FUNCTION_BLOCK FB_Carro_GRF_LD
// Transcripción del grafcet (GRF -> LD) [Usando células eléctricas de memoria]
VAR_INPUT
    ManiobrasTotales: UINT := 2;
    TiempoEspera: TIME := T#2S;
END_VAR
VAR_OUTPUT
    ManiobrasPendientes: UINT;
    TiempoPendiente: TIME;
END_VAR
VAR
    TiempoActual: TIME;
    
    // Variables propias del GRF
    S0x: BOOL := TRUE; // Etapa inicial
    S1x, S2x, S3x, S4x: BOOL; // Etapas no-iniciales
    t0, t1, t2, t3, t4, t4a: BOOL; // Transiciones
    S2t, S2_t: TIME; // S2.t y S2._t
    
    // Bloques funcionales
    FlancoPulsadorMarcha: R_TRIG;
    Intermitencia: FB_Blink;
    
    // Entradas
    i_PulsadorMarcha AT %I*: BOOL;
    i_FinalCarreraIzquierda AT %I*: BOOL := TRUE;
    i_FinalCarreraDerecha AT %I*: BOOL;
    
    // Salidas
    o_MarchaIzquierda AT %I*: BOOL;
    o_MarchaDerecha AT %I*: BOOL;
    o_LamparaMarcha AT %I*: BOOL;
END_VAR

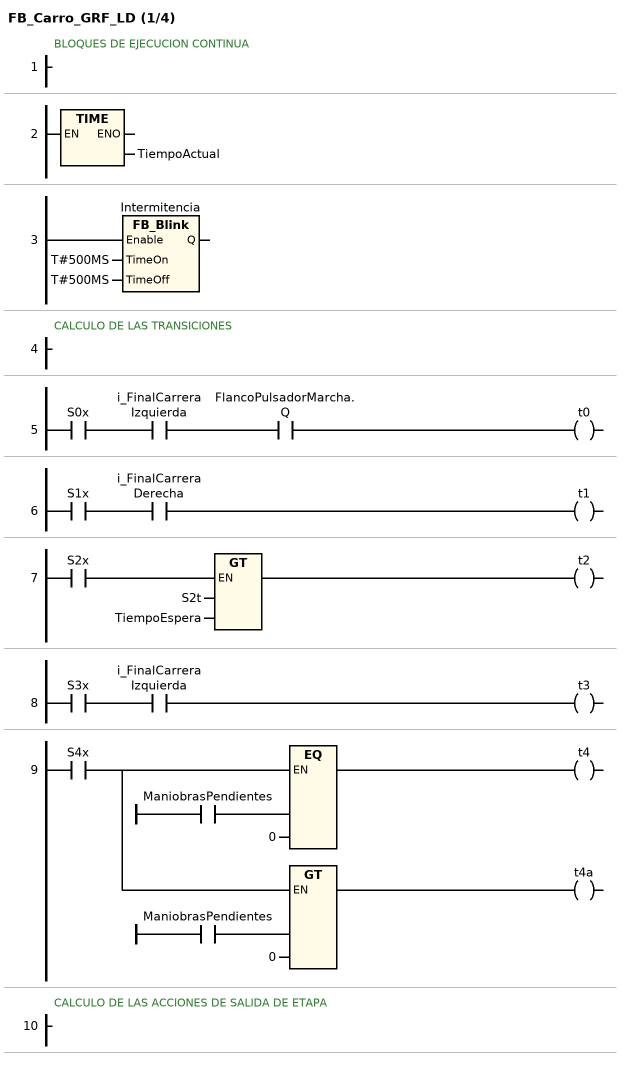
// NETWORK 1
// BLOQUES DE EJECUCION CONTINUA

// NETWORK 2
TiempoActual := TIME();

// NETWORK 3
Intermitencia(Enable := TRUE, TimeOn := T#500MS, TimeOff := T#500MS); // FB_Blink

// NETWORK 4
// CALCULO DE LAS TRANSICIONES

// NETWORK 5
t0 := S0x AND i_FinalCarreraIzquierda AND FlancoPulsadorMarcha.Q;

// NETWORK 6
t1 := S1x AND i_FinalCarreraDerecha;

// NETWORK 7
t2 := S2x AND S2t > TiempoEspera;

// NETWORK 8
t3 := S3x AND i_FinalCarreraIzquierda;

// NETWORK 9
t4 := S4x AND ManiobrasPendientes = 0;
t4a := S4x AND ManiobrasPendientes > 0;

// NETWORK 10
// CALCULO DE LAS ACCIONES DE SALIDA DE ETAPA

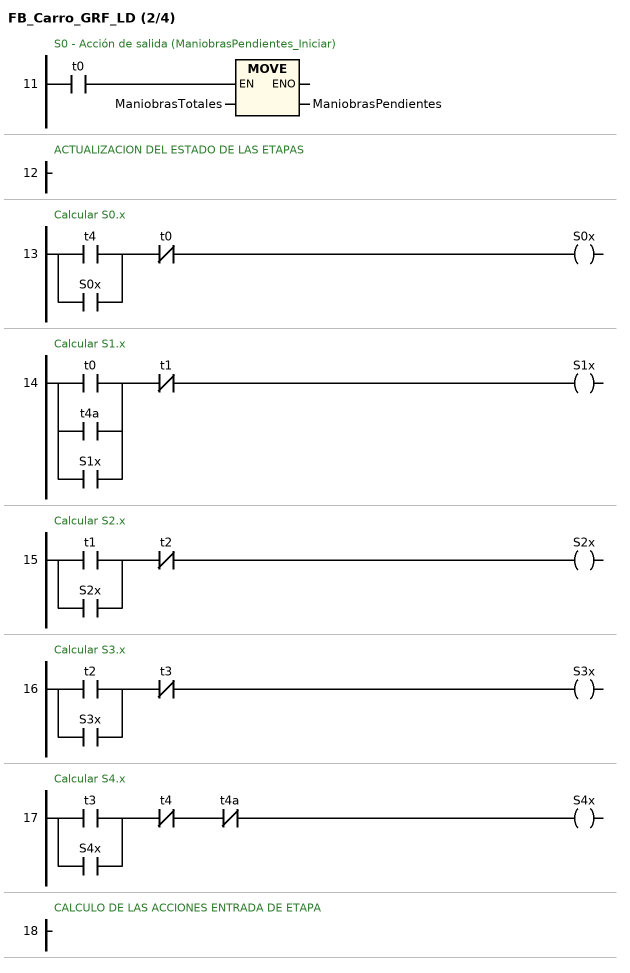
// NETWORK 11
// S0 - Acción de salida (ManiobrasPendientes_Iniciar)
IF t0 THEN ManiobrasPendientes := ManiobrasTotales; END_IF

// NETWORK 12
// ACTUALIZACION DEL ESTADO DE LAS ETAPAS

// NETWORK 13
// Calcular S0.x
S0x := (t4 OR S0x) AND NOT t0;

// NETWORK 14
// Calcular S1.x
S1x := (t0 OR t4a OR S1x) AND NOT t1;

// NETWORK 15
// Calcular S2.x
S2x := (t1 OR S2x) AND NOT t2;

// NETWORK 16
// Calcular S3.x
S3x := (t2 OR S3x) AND NOT t3;

// NETWORK 17
// Calcular S4.x
S4x := (t3 OR S4x) AND NOT t4 AND NOT t4a;

// NETWORK 18
// CALCULO DE LAS ACCIONES ENTRADA DE ETAPA

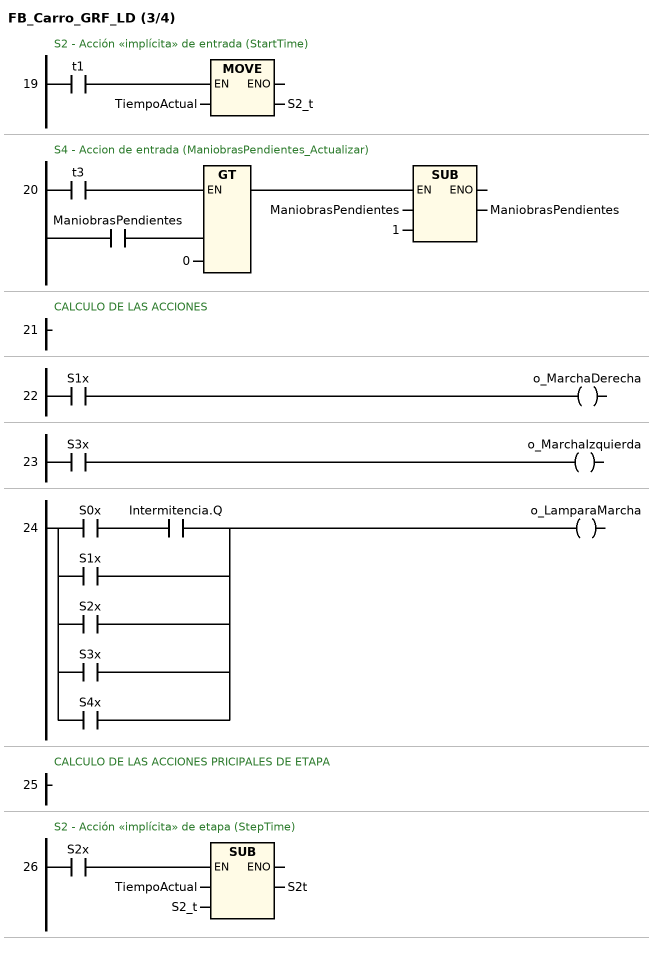
// NETWORK 19
// S2 - Acción «implícita» de entrada (StartTime)
IF t1 THEN S2_t := TiempoActual; END_IF

// NETWORK 20
// S4 - Accion de entrada (ManiobrasPendientes_Actualizar)
IF t3 AND ManiobrasPendientes > 0 THEN ManiobrasPendientes := ManiobrasPendientes - 1; END_IF

// NETWORK 21
// CALCULO DE LAS ACCIONES

// NETWORK 22
o_MarchaDerecha := S1x;

// NETWORK 23
o_MarchaIzquierda := S3x;

// NETWORK 24
o_LamparaMarcha := S0x AND Intermitencia.Q OR S1x OR S2x OR S3x OR S4x;

// NETWORK 25
// CALCULO DE LAS ACCIONES PRICIPALES DE ETAPA

// NETWORK 26
// S2 - Acción «implícita» de etapa (StepTime)
IF S2x THEN S2t := TiempoActual - S2_t; END_IF

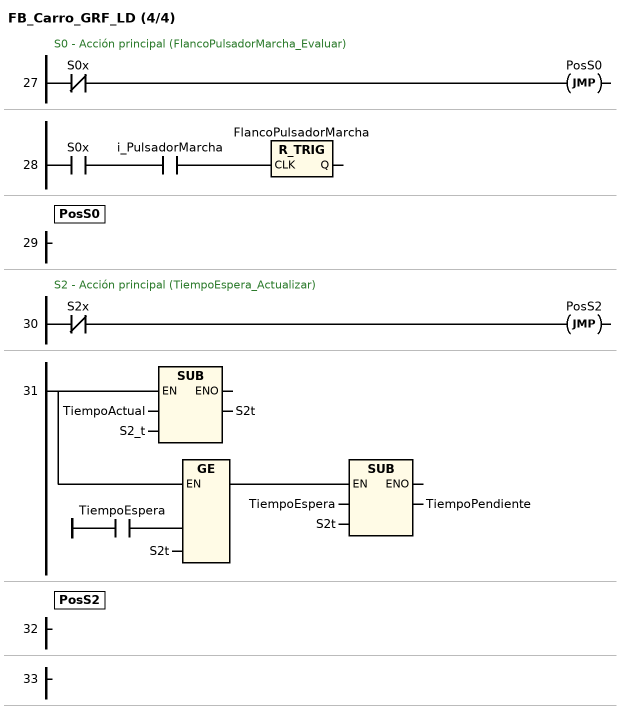
// NETWORK 27
// S0 - Acción principal (FlancoPulsadorMarcha_Evaluar)
IF NOT S0x THEN JMP PosS0; END_IF

// NETWORK 28
FlancoPulsadorMarcha(CLK := S0x AND i_PulsadorMarcha); // R_TRIG

// NETWORK 29
PosS0: ;

// NETWORK 30
// S2 - Acción principal (TiempoEspera_Actualizar)
IF NOT S2x THEN JMP PosS2; END_IF

// NETWORK 31
S2t := TiempoActual - S2_t;
IF TiempoEspera >= S2t THEN TiempoPendiente := TiempoEspera - S2t; END_IF

// NETWORK 32
PosS2: ;

// NETWORK 33

END_FUNCTION_BLOCK

(* stored: Version 1.1.0.1, ProductVersion 3.1.4024.16
   POU FB_Carro_GRF_LD: Id {49850c7a-a872-4ceb-b1dc-23d08810d361}, SpecialFunc None *)
